// TwinCAT 3 PLC project Main
// ProgramVersion: 3.1.4023.0
// libraries:
//   Tc2_Standard, * (Beckhoff Automation GmbH)
//   Tc2_System, * (Beckhoff Automation GmbH)
//   Tc2_Utilities, * (Beckhoff Automation GmbH)
//   Tc3_Module, * (Beckhoff Automation GmbH)
//   VisuDialogs, * (System)
//   VisuSymbols,3.5.10.0,System
// project tree:
//   Actuation Systems/Function Blocks/ BulkModulus.TcPOU (not stored), CraneAngle.TcPOU, DiscreteTimeIntegrator_Init.TcPOU (not stored), FWKinematics.TcPOU (not stored), HydraulicMotor.TcPOU, TimeIntegrator.TcPOU (not stored), HPU.TcPOU, CylinderMech.TcPOU, OrificeEquation.TcPOU (not stored), PressureGradient.TcPOU (not stored), Pump.TcPOU, ValveControlledCylinder.TcPOU (not stored), ValveDynamics.TcPOU
//   Actuation Systems/GVL/ G_ActuationSystems.TcGVL (not stored), Inputs.TcGVL (not stored), Work.TcGVL
//   Actuation Systems/Programs/ ActuationSystems.TcPOU
//   Functions/ Sign.TcPOU (not stored)
//   / GlobalTextList.TcGTLO (not stored), PlcTask.TcTTO (not stored), Visualization Manager.TcVMO (not stored)
//   Main Program/ MAIN.TcPOU (not stored), P_Joy.TcPOU (not stored)
//   Parameters/ Param.TcGVL, XboxControl.TcGVL (not stored)
//   Parameters/Structs/ Controller.TcDUT, ST_pValveControlledCylinder.TcDUT (not stored)
//   VISUs/ Visualization.TcVIS

// ---- Parameters/Structs/Controller.TcDUT
TYPE Controller :
STRUCT
	LeftJoystickX : INT;
	LeftJoystickY : INT;
	RightJoystickX : INT;
	RightJoystickY : INT;
	LeftTrigger : INT;
	RightTrigger : INT;
	LeftBumper : BOOL;
	RightBumper : BOOL;
	ButtonA : BOOL;
	ButtonB : BOOL;
	ButtonX : BOOL;
	ButtonY : BOOL;
	LeftThumb : BOOL;
	RightThumb : BOOL;
	Back : BOOL;
	Start : BOOL;
	DPadX : INT;
	DPadY : INT;
END_STRUCT
END_TYPE

// ---- Actuation Systems/GVL/Work.TcGVL
{attribute 'qualified_only'}
VAR_GLOBAL
	//To Unreal engine
	FpistonMainBoom : LREAL;
	FpistonKnuckleJib : LREAL;
	FpistonKingRotation : LREAL;
	
	
	//From Unreal engine
	VpistonMainBoom : LREAL;
	VpistonKnuckleJib : LREAL;
	VpistonKingRotation : LREAL;
	
	XpistonMainBoom : LREAL;
	XpistonKnuckleJib : LREAL;
	XpistonKingRotation : LREAL;
END_VAR

// ---- Parameters/Param.TcGVL
{attribute 'qualified_only'}
VAR_GLOBAL PERSISTENT
	pMainJibCylinder : ST_pValveControlledCylinder;				//Parameters for MainJibCylinder uses values from ST_pValveControlledCylinder
	pKnuckleJibCylinder : ST_pValveControlledCylinder; 			//Parameters for KnuckleJib uses values from ST_pValveControlledCylinderv
	pKingRotationCylinder : ST_pValveControlledCylinder;        //Parameters for KingRotation uses values from ST_pValveControlledCylinderv
END_VAR

// ---- Actuation Systems/Function Blocks/CraneAngle.TcPOU
FUNCTION_BLOCK CraneAngle
VAR_INPUT
	par : ST_pValveControlledCylinder;
	a : LREAL;
	b : LREAL;
	c : LREAL;
END_VAR
VAR_OUTPUT
	thetaAngle : LREAL;
END_VAR
VAR
    thetaAngleRad : LREAL;
	thetaAngleDeg : LREAL;
END_VAR


//Angle A joint 1 and joint 2
//thetaAngle := ACOS( (EXPT(b,2) + EXPT(c,2) - EXPT(a,2) ) / ((2) * b * c));

//To make it into degrees if i need that:
thetaAngleDeg := thetaAngle*(180/par.pi);

END_FUNCTION_BLOCK

// ---- Actuation Systems/Function Blocks/HydraulicMotor.TcPOU
FUNCTION_BLOCK HydraulicMotor
VAR_INPUT
	par : ST_pValveControlledCylinder;
	PressureIn : LREAL;
	PressureOut : LREAL;
END_VAR
VAR_OUTPUT
	Torque : LREAL;
END_VAR
VAR
	dpsum : LREAL;					//[pa]
	Dm : LREAL := 189;				//[cm^3/Rev]
	nhm : LREAL := 0.9;			//[-]
END_VAR

//For controlling the king joint, aka rotation of the whole crane horisontally
//dpsum = (PressureIn - PressureOut);

dpsum := (PressureIn - PressureOut);

Torque := ( dpsum * Dm * nhm * EXPT(10,(-6))) / (2 * par.pi);

END_FUNCTION_BLOCK

// ---- Actuation Systems/Function Blocks/HPU.TcPOU
FUNCTION_BLOCK HPU
VAR_INPUT
	par : ST_pValveControlledCylinder;
END_VAR
VAR_OUTPUT
	TankPressure : LREAL;
	SupplyPressure : LREAL;
END_VAR
VAR
	//Pump
	fbPump : Pump;
	PumpTorque : LREAL;
	PumpFlowRate : LREAL;
END_VAR


//Pump
fbPump(
MotorSpeedRPM := 413.2,
PumpDisplacement := 10.6E-6,
DeltaMaxPressure := 250.0E5,
PumpTorque => PumpTorque,
PumpFlowRate => PumpFlowRate
);

TankPressure := 1.2E5;  			//[Pa]
SupplyPressure := 250E5; 			//[Pa]

G_ActuationSystems.ReturnPressure := TankPressure;
G_ActuationSystems.SupplyPressure := SupplyPressure;

END_FUNCTION_BLOCK

// ---- Actuation Systems/Function Blocks/Pump.TcPOU
FUNCTION_BLOCK Pump
VAR_INPUT
	MotorSpeedRPM: LREAL;
	PumpDisplacement: LREAL;
	DeltaMaxPressure: LREAL;
	PistonVelocity4Pump : LREAL;
	par : ST_pValveControlledCylinder;
END_VAR
VAR_OUTPUT
	PumpTorque: LREAL;
	PumpFlowRate: LREAL;
END_VAR
VAR

	// Trying to make the system go towards a certain set xpos
(*	xDeviation : LREAL;
	xSet : LREAL := 0.7;
	vDeviation : LREAL;
	fbVelocity : DiscreteIntegrator;
	vDeviationPre : LREAL;
	*)
END_VAR


PumpTorque := (DeltaMaxPressure * PumpDisplacement) * 15915.494309189535;

PumpFlowRate := (PumpDisplacement * MotorSpeedRPM) * 1000.0;

END_FUNCTION_BLOCK

// ---- Actuation Systems/Function Blocks/CylinderMech.TcPOU
FUNCTION_BLOCK CylinderMech
VAR_INPUT
	//PressureBoreSide : LREAL;
	//PressureRodSide : LREAL;
	param : ST_pValveControlledCylinder;
	F_Hydraulic : LREAL;
END_VAR
VAR_OUTPUT
	PistonAcceleration: LREAL;
	PistonVelocity : LREAL;
	PistonPosition : LREAL;
	F_Piston : LREAL;
END_VAR
VAR
	ssMethodType : SINT := 1; 
	fbPistonVelocity : DiscreteTimeIntegrator_Init;
	fbPistonPosition : DiscreteTimeIntegrator_Init;
	y_tmp : LREAL;
	SpringContactCoefficient : LREAL;
	DamperContactCoefficient : LREAL;
	F_Upper_Stroke_Limit : LREAL;
	F_Lower_Stroke_Limit : LREAL;
	F_Stribeck_Friction : LREAL;
	AbsPosition: LREAL;
END_VAR

// Upper Stroke Limit Contact Force [N] //
IF PistonPosition >= param.xMax THEN 
	SpringContactCoefficient := param.cyl_k_end;
ELSIF PistonPosition < param.xMax THEN 
	SpringContactCoefficient := 0;
END_IF;	

IF PistonPosition >= param.xMax THEN 
	DamperContactCoefficient := param.cyl_c_end;
ELSIF PistonPosition < param.xMax THEN 
	DamperContactCoefficient := 0;
END_IF;	

F_Upper_Stroke_Limit := ((PistonPosition - param.xMax) * SpringContactCoefficient) + (DamperContactCoefficient * PistonVelocity);



//// Lower Stroke Limit Contact Force [N] //
IF PistonPosition > 0 THEN 
	SpringContactCoefficient := 0;
ELSIF PistonPosition <= 0 THEN 
	SpringContactCoefficient := param.cyl_k_end;
END_IF;	

IF PistonPosition > 0 THEN 
	DamperContactCoefficient := 0;
ELSIF PistonPosition <= 0 THEN 
	DamperContactCoefficient := param.cyl_c_end;
END_IF;	

AbsPosition := ABS(PistonPosition);
F_Lower_Stroke_Limit := (SpringContactCoefficient * AbsPosition) + (DamperContactCoefficient * (-1) * PistonVelocity);



//// Stribeck Friction Force [N] //
//y_tmp := EXP((PistonVelocity * param.FrictionForceApproximationConstant) * 2.0);
//y_tmp := (y_tmp - 1.0) / (y_tmp + 1.0);
//F_Stribeck_Friction := (((EXP(( -(PistonVelocity * y_tmp)) / param.StaticFrictionTimeConstant) * ABS(param.StaticFrictionForce)) + param.ColoumbFriction) * y_tmp) + (PistonVelocity * param.ViscousFrictionCoefficient);


/// Piston Force Total [N] ///
F_Piston := ( (F_Hydraulic - F_Upper_Stroke_Limit + F_Lower_Stroke_Limit - F_Stribeck_Friction) ) * 4;


// Piston Acceleration [m/s^2]
PistonAcceleration := (F_Piston - param.ExternalForce) / param.EffectiveMass;

PistonVelocity := Work.VpistonMainBoom; 	//From Unreal engine
PistonPosition := Work.XpistonMainBoom;		//From Unreal engine

//fbPistonVelocity(
//	ssMethodType := ssMethodType,
//	tCycle := param.tCycle,
//	In := PistonAcceleration,
//	Init := param.v0,
//	minOut := -param.vMax,
//	maxOut := param.vMax,
//	Out => PistonVelocity
//	);

//fbPistonPosition(
//	ssMethodType := ssMethodType,
//	tCycle := param.tCycle,
//	In := PistonVelocity,
//	Init := param.x0,
//	minOut := -5000,
//	maxOut := param.xMax+5000,
//	Out => PistonPosition
//	);

//IF PistonPosition >= param.xMax THEN 
//	PistonPosition := param.xMax;
//ELSIF PistonPosition <= 0 THEN 
//	PistonPosition := 0;
//END_IF;

END_FUNCTION_BLOCK

// ---- Actuation Systems/Function Blocks/ValveDynamics.TcPOU
FUNCTION_BLOCK ValveDynamics
VAR_INPUT
	udcv_IN : LREAL;
	wn : LREAL := 30.0;
	dr : LREAL := 0.7;
END_VAR
VAR_OUTPUT
	DynamicValve : LREAL;
END_VAR
VAR
	fDeltaTime : LREAL := 0.001;
	fAcceleration : LREAL;
	fbVelocity : TimeIntegrator := (fInit := 0.0);
	fbPosition : TimeIntegrator := (fInit := 0.0);
	a : LREAL;
	b : LREAL;
END_VAR
VAR CONSTANT
END_VAR

//Timer := Timer + 0.001;

////Valve opening signal is sent through this
//DynamicValve := cst1*EXP(-21*Timer)*SIN(cst2*Timer);

IF (wn = 0.0) THEN
	RETURN;
END_IF

a := 1/EXPT(wn, 2.0);
b := dr/wn;

fAcceleration := (udcv_IN - 2*fbVelocity.fOut*b - fbPosition.fOut)/a;

fbVelocity(
	fIn := fAcceleration,
	fStepTime := fDeltaTime,
);

fbPosition(
	fIn := fbVelocity.fOut,
	fStepTime := fDeltaTime,
	bEnableLimits := TRUE,
	fMinVal := -1.0,
	fMaxVal := 1.0,
	fOut => DynamicValve
);

END_FUNCTION_BLOCK

// ---- Actuation Systems/Programs/ActuationSystems.TcPOU
PROGRAM ActuationSystems
VAR
fbMainJibCylinderHyd : ValveControlledCylinder;
fbKnuckleJibCylinderHyd : ValveControlledCylinder;
fbKingRotationCylinderHyd : ValveControlledCylinder;
//HydraulicCylinder
fbMainJibCylinderMech : CylinderMech;
fbKnuckleJibCylinderMech : CylinderMech;
fbkingRotationCylinderMech : CylinderMech;

fbFWKinematics : FWKinematics;
fbHPU : HPU;
END_VAR

fbHPU(
);

fbFWKinematics(
	L1 := 4.543126+1.097+1.000,  												//[m]
	L2 := 0,																	//[m]
	L3 := 17.939373,															//[m]
	L4 := 9.548784,																//[m]
	thetaMainBoom := ActuationSystems.fbKnuckleJibCylinderHyd.AngleJoint,		//[rad]
	thetaKnuckleBoom := ActuationSystems.fbMainJibCylinderHyd.AngleJoint, 		//[rad]
	thetaSlew := 0																//[rad]
);

//Hyd Model for MainJibCylinder
fbMainJibCylinderHyd(
	uDcvEnable := Inputs.uDcvEnableMainJib,
	uDcv := Inputs.uDcvMainJib,	
	ReturnPressure := G_ActuationSystems.ReturnPressure,
	SupplyPressure := G_ActuationSystems.SupplyPressure,
	par := Param.pMainJibCylinder,
	xPiston := fbMainJibCylinderMech.PistonPosition,
	vPiston := fbMainJibCylinderMech.PistonVelocity,
);
//Hyd Model for KnuckleJibCylinder
fbKnuckleJibCylinderHyd(
	uDcvEnable := Inputs.uDcvEnableKnuckleJib,
	uDcv := Inputs.uDcvKnuckleJib,	
	ReturnPressure := G_ActuationSystems.ReturnPressure,
	SupplyPressure := G_ActuationSystems.SupplyPressure,
	par := Param.pKnuckleJibCylinder,
	xPiston := fbKnuckleJibCylinderMech.PistonPosition,
	vPiston := fbKnuckleJibCylinderMech.PistonVelocity,
);
//Hyd Model for KingRotationCylinder
fbKingRotationCylinderHyd(
	uDcvEnable := Inputs.uDcvEnableKingRotation,
	uDcv := Inputs.uDcvKingRotation,	
	ReturnPressure := G_ActuationSystems.ReturnPressure,
	SupplyPressure := G_ActuationSystems.SupplyPressure,
	par := Param.pMainJibCylinder,
	xPiston := fbkingRotationCylinderMech.PistonPosition,
	vPiston := fbkingRotationCylinderMech.PistonVelocity,
);


//Temp Mechanical Model for MainJibCylinder
fbMainJibCylinderMech(
	F_Hydraulic := fbMainJibCylinderHyd.F_Hydraulic,
	param := Param.pMainJibCylinder,
	F_Piston => Work.FpistonMainBoom
);	
//Temp Mechanical Model for KnuckleJibCylinder
fbKnuckleJibCylinderMech(
	F_Hydraulic := fbKnuckleJibCylinderHyd.F_Hydraulic,
	param := Param.pKnuckleJibCylinder,
	F_Piston => Work.FpistonKnuckleJib
);	
//Temp Mechanical Model for KingRotationCylinder
fbkingRotationCylinderMech(
	F_Hydraulic := fbKingRotationCylinderHyd.F_Hydraulic,
	param := Param.pKingRotationCylinder,
	F_Piston => Work.FpistonKingRotation
);

END_PROGRAM

// ---- VISUs/Visualization.TcVIS
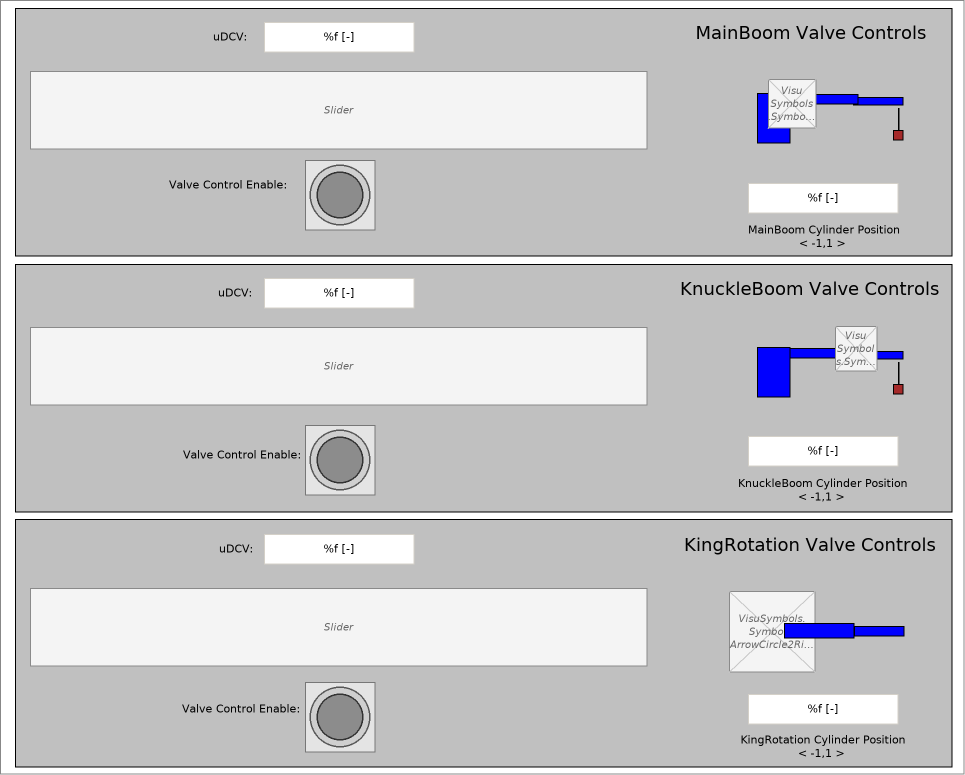
VISUALIZATION Visualization  // 965x775
    RoundedRectangle (15,519 937x248)
    RoundedRectangle (15,264 937x248)
    RoundedRectangle (15,8 937x248)
    Slider (30,71 617x78), variable: Inputs.uDcvMainJib, scale -1..1
    PushSwitchLed (305,160 70x70), variable: Inputs.uDcvEnableMainJib, behaviour: TOGGLE, style: Switch-PushSwitchLed-Gray
    Textfield (264,22 150x30), "%f [-]", text variable: Inputs.uDcvMainJib
        OnMouseClick: write the text variable via Default, min -1, max 1
    Label (197,22 66x30), "uDCV:"
    Label (137,170 182x30), "Valve Control Enable:"
    Slider (30,327 617x78), variable: Inputs.uDcvKnuckleJib, scale -1..1
    PushSwitchLed (305,425 70x70), variable: Inputs.uDcvEnableKnuckleJib, behaviour: TOGGLE, style: Switch-PushSwitchLed-Gray
    Textfield (264,278 150x30), "%f [-]", text variable: Inputs.uDcvKnuckleJib
        OnMouseClick: write the text variable via Default, min -1, max 1
    Label (202,278 66x30), "uDCV:"
    Label (151,440 182x30), "Valve Control Enable:"
    Label (676,18 270x30), "MainBoom Valve Controls"
    Label (675,274 270x30), "KnuckleBoom Valve Controls"
    Slider (30,588 617x78), variable: Inputs.uDcvKingRotation, scale -1..1
    PushSwitchLed (305,682 70x70), variable: Inputs.uDcvEnableKingRotation, behaviour: TOGGLE, style: Switch-PushSwitchLed-Gray
    Textfield (264,534 150x30), "%f [-]", text variable: Inputs.uDcvKingRotation
        OnMouseClick: write the text variable via Default, min -1, max 1
    Label (203,534 66x30), "uDCV:"
    Label (150,694 182x30), "Valve Control Enable:"
    Label (675,530 270x30), "KingRotation Valve Controls"
    Ellipse (757,616 30x30)
    Image (729,591 86x81), angle 320, image: VisuSymbols.Symbols.ArrowCircle2RightRightLeft
    Rectangle (854,626 50x10)
    Rectangle (784,623 70x15)
    Rectangle (887,373 22x1), angle 270
    Rectangle (853,351 50x8), angle 203
    Rectangle (788,348 70x10), angle 349
    Rectangle (757,347 33x50)
    Rectangle (893,384 10x10)
    Rectangle (757,93 33x50)
    Rectangle (887,119 22x1), angle 270
    Rectangle (853,97 50x8), angle 203
    Rectangle (788,94 70x10), angle 349
    Rectangle (893,130 10x10)
    Image (768,79 48x49), angle 345, image: VisuSymbols.Symbols.ArrowCircle2LeftUpDown
    Image (835,326 42x45), angle 10, image: VisuSymbols.Symbols.ArrowCircle2LeftUpDown
    Textfield (748,183 150x30), "%f [-]", text variable: ActuationSystems.fbMainJibCylinderHyd.xPiston
        OnMouseClick: write the text variable via Default, min -1, max 1
    Textfield (748,436 150x30), "%f [-]", text variable: ActuationSystems.fbKnuckleJibCylinderHyd.xPiston
        OnMouseClick: write the text variable via Default, min -1, max 1
    Textfield (748,694 150x30), "%f [-]", text variable: ActuationSystems.fbKingRotationCylinderHyd.xPiston
        OnMouseClick: write the text variable via Default, min -1, max 1
    Label (682,460 282x60), "KnuckleBoom Cylinder Position < -1,1 >"
    Label (682,718 282x57), "KingRotation Cylinder Position < -1,1 >"
    Label (683,206 282x61), "MainBoom Cylinder Position < -1,1 >"
END_VISUALIZATION
